// TIA Portal V20 export
DATA_BLOCK "G2_上传"   // DB2
{ S7_Optimized_Access := 'FALSE' }
   VAR
      位1 : Bool;
      位2 : Bool;
      位3 : Bool;
      位4 : Bool;
      位5 : Bool;
      位6 : Bool;
      位7 : Bool;
      位8 : Bool;
      位9 : Bool;
      位10 : Bool;
      位11 : Bool;
      位12 : Bool;
      位13 : Bool;
      位14 : Bool;
      位15 : Bool;
      位16 : Bool;
      位17 : Bool;
      位18 : Bool;
      位19 : Bool;
      位20 : Bool;
      位21 : Bool;
      位22 : Bool;
      位23 : Bool;
      位24 : Bool;
      位25 : Bool;
      位26 : Bool;
      位27 : Bool;
      位28 : Bool;
      位29 : Bool;
      位30 : Bool;
      整型1 : Int;
      整型2 : Int;
      整型3 : Int;
      整型4 : Int;
      整型5 : Int;
      整型6 : Int;
      整型7 : Int;
      整型8 : Int;
      整型9 : Int;
      整型10 : Int;
      浮点数1 : Real;
      浮点数2 : Real;
      浮点数3 : Real;
      浮点数4 : Real;
      浮点数5 : Real;
      浮点数6 : Real;
      浮点数7 : Real;
      浮点数8 : Real;
      浮点数9 : Real;
      浮点数10 : Real;
      浮点数11 : Real;
      浮点数12 : Real;
      浮点数13 : Real;
      浮点数14 : Real;
      浮点数15 : Real;
      浮点数16 : Real;
      浮点数17 : Real;
      浮点数18 : Real;
      浮点数19 : Real;
   END_VAR
BEGIN
END_DATA_BLOCK
